# EPICS substitutions: Galil-test/GalilTestApp/Db/asynRecord.substitutions
file "$(GALIL)/GalilSup/Db/asynRecord.template"
{
 pattern
 { P		, R		, PORT		, ADDR	, OMAX	, IMAX	}
 { Test		, "{DMC:1}Asyn"	, Galil		, 0	, 80	, 80	}
}
